INTERFACE I_SnappySetupDefaultsOrRpc

METHOD UseDefaults : I_SnappySetupConfigTestFrameWork
VAR_INPUT
END_VAR
END_METHOD

METHOD UseRpcProxy : I_SnappySetupConfigSerializer
VAR_INPUT
	itfRpcProxy	: I_RpcProxy;
END_VAR
END_METHOD

END_INTERFACE

(* stored: Version 1.1.0.1, ProductVersion 3.1.4026.18
   Itf I_SnappySetupDefaultsOrRpc: Id {fb50fff0-a471-4ada-a732-1db0d4ca1261}
   Method UseDefaults: Id {cfd5f940-2d41-4f19-ab6f-fcbd0edd34e0}
   Method UseRpcProxy: Id {f22ce6f3-1b8c-4781-b95d-49cbf5611232} *)
